// TIA Portal V20 export
TYPE "typeEm4Monitoring"
// stored: Access Published, Namespace Unit1
   STRUCT
      cmStatus { ExternalWritable := 'False'} : "Unit1.typeEm4MonitoringCmStatus";
      JobStatus { ExternalWritable := 'False'} : "Unit1.typeEm4MonitoringJobStatus";
      UserDefine { ExternalWritable := 'False'} : "Unit1.typeEm4MonitoringUserDefine";
   END_STRUCT;
END_TYPE
